Fanuc TP program (LS listing): RSR0001.LS

/PROG  RSR0001
/ATTR
OWNER		= MNEDITOR;
COMMENT		= "RSR1 -> KMX_PLAY";
PROG_SIZE	= 0;
CREATE		= DATE 00-00-00  TIME 00:00:00;
MODIFIED	= DATE 00-00-00  TIME 00:00:00;
FILE_NAME	= ;
VERSION		= 0;
LINE_COUNT	= 1;
MEMORY_SIZE	= 0;
PROTECT		= READ_WRITE;
TCD:  STACK_SIZE	= 0,
      TASK_PRIORITY	= 50,
      TIME_SLICE	= 0,
      BUSY_LAMP_OFF	= 0,
      ABORT_REQUEST	= 0,
      PAUSE_REQUEST	= 0;
DEFAULT_GROUP	= 1,*,*,*,*;
CONTROL_CODE	= 00000000 00000000;
/APPL
/MN
  1:  CALL KMX_PLAY    ;
/POS
/END
